// TwinCAT 3 PLC project EtherCatDevice
// Title: EtherCatDevice
// Company: NewEngineer
// Author: https://github.com/phucpha
// ProjectVersion: 0.0.0.2
// Description: this is library use for Device conmunicate by EtherCat without requrire special license.
// ProgramVersion: 3.1.4024.0
// libraries:
//   Tc2_Math, * (Beckhoff Automation GmbH)
//   Tc2_Standard, * (Beckhoff Automation GmbH)
//   Tc2_System, * (Beckhoff Automation GmbH)
//   Tc3_Module, * (Beckhoff Automation GmbH)
//   VisuDialogs, * (System)
//   VisuSymbols,3.5.10.0,System
// project tree:
//   DUTs/Robots/Mitsubishi/CR800/EtherCAT Registers/ ST_CR800EthercatData.TcDUT (not stored)
//   DUTs/Robots/Mitsubishi/CR800/ E_CR800Error.TcDUT (not stored), ST_CR800UserDefinedArea.TcDUT (not stored)
//   DUTs/Robots/Mitsubishi/CR800/StateMachine/ E_CR800State.TcDUT (not stored), E_CR800StateAborting.TcDUT (not stored), E_CR800StateCommandExchange.TcDUT (not stored), E_CR800StateCyclePausing.TcDUT (not stored), E_CR800StateCycleStopping.TcDUT (not stored), E_CR800StateDoingRequest.TcDUT (not stored), E_CR800StateHoming.TcDUT (not stored), E_CR800StateInitializing.TcDUT (not stored), E_CR800StateSendPosition.TcDUT (not stored)
//   DUTs/Robots/Mitsubishi/ E_RobotActions.TcDUT (not stored), E_RobotSystemActions.TcDUT (not stored)
//   DUTs/Visu/ ST_VisuCtrlRobotFrame.TcDUT
//   / GlobalTextList.TcGTLO, PlcTask.TcTTO, Visualization Manager.TcVMO (not stored)
//   POUs/Robots/Mitsubishi/ FB_CR800EtherCAT.TcPOU (not stored), I_CR800EtherCAT.TcIO (not stored)
//   Version/ Global_Version.TcGVL
//   VISUs/Image Polls/ IPRobots.TcIPO (not stored)
//   VISUs/Pages/ PageManualRobots.TcVIS
//   VISUs/Single/ SingleRobot.TcVIS
//   VISUs/Text Lists/ TL_ModeSwitchState.TcTLO, TL_SingleRobotState.TcTLO
// real-time tasks:
//   TASK PlcTask: cycle T#10ms, priority 20, ADS port 350

CONFIGURATION EtherCatDevice
    RESOURCE PLC ON TwinCAT3
        TASK PlcTask(INTERVAL := T#10ms, PRIORITY := 20);
    END_RESOURCE
END_CONFIGURATION

// ---- DUTs/Visu/ST_VisuCtrlRobotFrame.TcDUT
TYPE ST_VisuCtrlRobotFrame :
STRUCT
	sName 						: STRING := 'Unknown';
	btnInit						: BOOL;				(*  *)
	btnAbort					: BOOL;				(*  *)
	btnErrorReset				: BOOL;				(*  *)
	btnControllerReset			: BOOL;				(*  *)
	btnBatteryReset				: BOOL;				(*  *)
	btnGoHome 					: BOOL;				(*  *)
	btnDoAction	 				: BOOL;				(*  *)
	btnUpdateRecipes			: BOOL;				(*  *)
	btnGoAuto 					: BOOL;				(*  *)
	btnCyclePause				: BOOL;				(*  *)
	btnCycleStop				: BOOL;				(*  *)
	btnRestoreCycle 			: BOOL;				(*  *)
	btnRestoreAuto	 			: BOOL;				(*  *)
	btnModeSwitch	 			: BOOL;				(*  *)
	bModeSwitchButtonDisabled	: BOOL;
	
	bError						: BOOL;				(*  *)
	bInit						: BOOL;	
	bPowerOn					: BOOL;	
	bBatteryLow					: BOOL;	
	bIsHomed					: BOOL;
	bServoOn					: BOOL;				(*  *)
	bServoOff 					: BOOL;
	bStarted					: BOOL;
	bStopped					: BOOL;				(*  *)
	bPaused						: BOOL;
	bUninitialized				: BOOL;
	bDoAction					: BOOL;
	bAutoButtonDisable			: BOOL;	
	bActionButtonDisable		: BOOL;	
	bHomeButtonDisable 			: BOOL;
	bPausingButtonDisable 		: BOOL;
	bRestoreCycleButtonDisable  : BOOL;
	bStoppingButtonDisable	    : BOOL;
	bRestoreAutoButtonDisable   : BOOL;
	bInitButtonDisable			: BOOL;
	bModeSwitchState			: BOOL;
	
	sErrorDescription			: STRING;			(*  *)
	iActionNumber				: UINT := 51;		(*  *)
	iOverride					: USINT := 100;
	sStateDescription			: STRING;			(*  *)
	
	sRobotImage					: STRING;			(*  *)
	eRobotState					: E_CR800State;		(*  *)
END_STRUCT
END_TYPE

// ---- Version/Global_Version.TcGVL
{attribute 'TcGenerated'}
{attribute 'no-analysis'}
{attribute 'linkalways'}
// This function has been automatically generated from the project information.
VAR_GLOBAL CONSTANT
	{attribute 'const_non_replaced'}
	stLibVersion_EtherCatDevice : ST_LibVersion := (iMajor := 0, iMinor := 0, iBuild := 0, iRevision := 2, nFlags := 0, sVersion := '0.0.0.2');
END_VAR

// ---- GlobalTextList.TcGTLO
TEXTLIST GlobalTextList
  224 = '%2d'
  331 = '%d'
  976 = '%s'
  2051 = '/'
  887 = 'Abort'
  3798 = 'Action number:'
  427 = 'Auto mode'
  2272 = 'Battery low'
  662 = 'Battery reset'
  1072 = 'Commands'
  1156 = 'Controller'
  2043 = 'Cycle pause'
  3558 = 'Cycle restore'
  1468 = 'Error'
  1738 = 'Error: %s'
  66 = 'Go home'
  1505 = 'Homed'
  371 = 'Initialize'
  1488 = 'Initialized'
  729 = 'Mode switch'
  1606 = 'Next'
  725 = 'Paused'
  731 = 'Powered on'
  1825 = 'Previous'
  316 = 'Program'
  3075 = 'Reset'
  951 = 'Robots'
  2402 = 'Servo off'
  772 = 'Servo on'
  450 = 'Start'
  3789 = 'Started'
  1037 = 'State: %s'
  895 = 'Status'
  1093 = 'Stopped'
END_TEXTLIST

// ---- VISUs/Pages/PageManualRobots.TcVIS
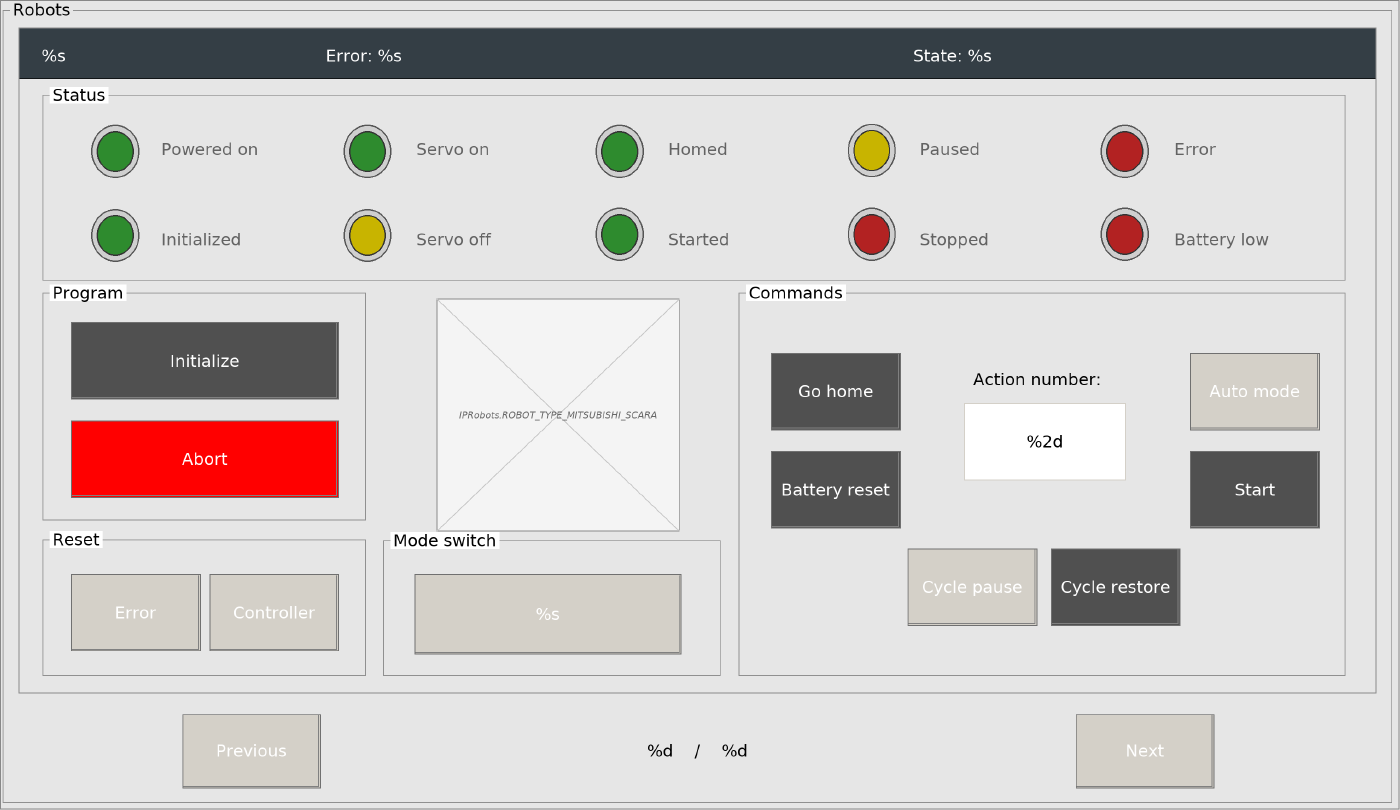
VISUALIZATION PageManualRobots  // 1520x880
VAR_IN_OUT
	btnPrevious			: BOOL;
	btnNext				: BOOL;
	bPreviousInvisible	: BOOL;
	bNextInvisible		: BOOL;
	stRobotEmpty		: ARRAY[1..1] OF BOOL;
	stRobot				: ARRAY[1..1] OF ST_VisuCtrlRobotFrame;
	iRobotSelectedPageIndex	: USINT;
	iRobotTotalPageIndex 	: USINT;
	
END_VAR
    GroupBox (3,3 1508x869), "Robots"
        Button (195,773 150x80), "Previous", invisible if: bPreviousInvisible
            tap btnPrevious
        Button (1165,773 150x80), "Next", invisible if: bNextInvisible
            tap btnNext
        Frame (17,27 1474x723), invisible if: stRobotEmpty[1]
            shows SingleRobot(stRobot := stRobot[1])
        Rectangle (689,788 130x50), "/"
        Rectangle (689,788 50x50), "%d", text variable: iRobotSelectedPageIndex+1
        Rectangle (770,788 50x50), "%d", text variable: iRobotTotalPageIndex+1
END_VISUALIZATION

// ---- VISUs/Single/SingleRobot.TcVIS
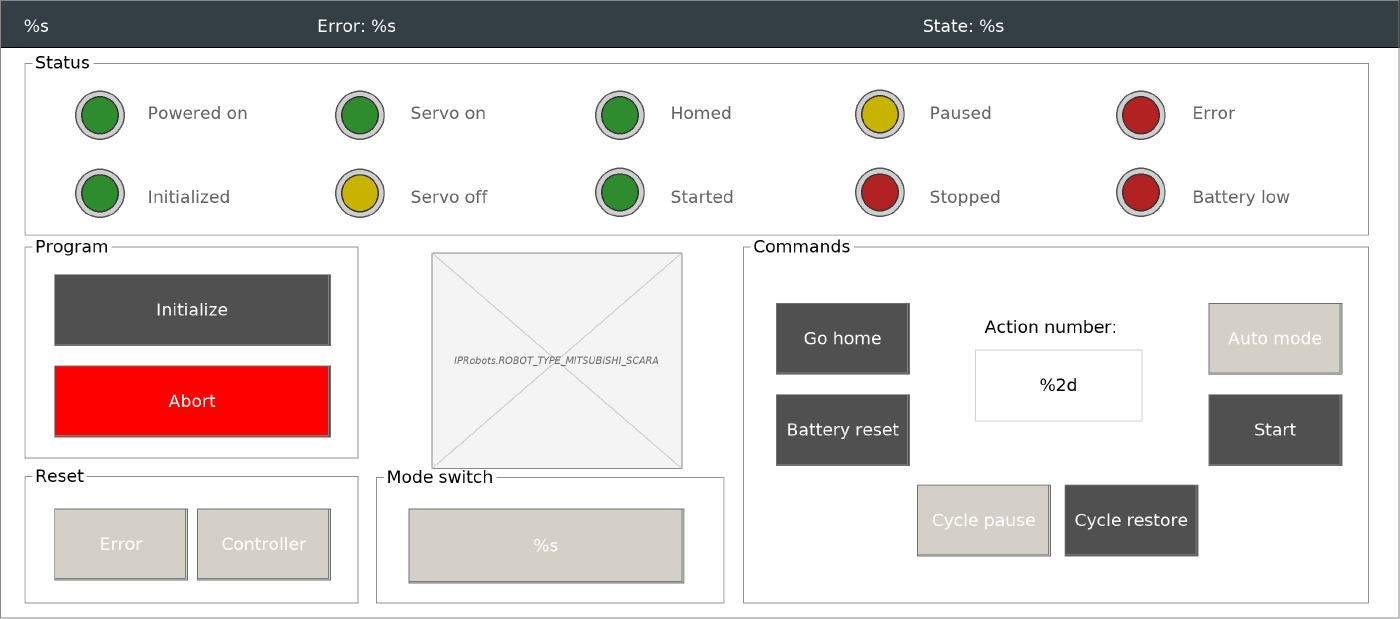
VISUALIZATION SingleRobot  // 1470x650
VAR_IN_OUT
	stRobot		: ST_VisuCtrlRobotFrame;
END_VAR
    Rectangle (0,0 1470x50)
    Textfield (22,10 296x35), "%s", text variable: stRobot.sName
    Textfield (966,10 498x35), "State: %s", text list: 'TL_SingleRobotState', text index: stRobot.eRobotState
    Textfield (330,10 628x35), "Error: %s", text variable: stRobot.sErrorDescription
    Image (453,265 263x227), image: IPRobots.ROBOT_TYPE_MITSUBISHI_SCARA
        p84334746: stRobot.sRobotImage
    GroupBox (26,58 1411x189), "Status"
        Lamp1 (595,33 60x60), variable: stRobot.bIsHomed, style: Lamp-Lamp1-Green
        Lamp1 (595,114 60x60), variable: stRobot.bStarted, style: Lamp-Lamp1-Green
        Rectangle (675,37 150x48), "Homed"
        Rectangle (675,125 150x48), "Started"
        Lamp1 (1142,114 60x60), variable: stRobot.bBatteryLow, style: Lamp-Lamp1-Red
        Rectangle (1223,125 150x48), "Battery low"
        Lamp1 (1142,33 60x60), variable: stRobot.bError, style: Lamp-Lamp1-Red
        Rectangle (1223,37 150x48), "Error"
        Lamp1 (49,33 60x60), variable: stRobot.bPowerOn, style: Lamp-Lamp1-Green
        Lamp1 (49,115 60x60), variable: stRobot.bInit, style: Lamp-Lamp1-Green
        Rectangle (126,37 150x48), "Powered on"
        Rectangle (126,125 150x48), "Initialized"
        Rectangle (402,37 150x48), "Servo on"
        Rectangle (402,125 150x48), "Servo off"
        Lamp1 (322,33 60x60), variable: stRobot.bServoOn, style: Lamp-Lamp1-Green
        Lamp1 (322,115 60x60), variable: stRobot.bServoOff, style: Lamp-Lamp1-Yellow
        Rectangle (947,37 150x48), "Paused"
        Rectangle (947,125 150x48), "Stopped"
        Lamp1 (868,32 60x60), variable: stRobot.bPaused, style: Lamp-Lamp1-Yellow
        Lamp1 (868,114 60x60), variable: stRobot.bStopped, style: Lamp-Lamp1-Red
    GroupBox (26,251 350x230), "Program"
        Button (31,37 290x75), "Initialize", input disabled if: stRobot.bInitButtonDisable
            tap stRobot.btnInit
        Button (31,133 290x75), "Abort", input disabled if: stRobot.bUninitialized
            tap stRobot.btnAbort
    GroupBox (26,492 350x141), "Reset"
        Button (31,42 140x75), "Error"
            tap stRobot.btnErrorReset
        Button (181,42 140x75), "Controller"
            tap stRobot.btnControllerReset
    GroupBox (780,251 657x382), "Commands"
        Button (489,163 140x75), "Start", input disabled if: stRobot.bActionButtonDisable
            tap stRobot.btnDoAction
        Button (35,67 140x75), "Go home", input disabled if: stRobot.bHomeButtonDisable
            tap stRobot.btnGoHome
        Button (489,67 140x75), "Auto mode", input disabled if: stRobot.bAutoButtonDisable
            tap stRobot.btnGoAuto
        Button (35,163 140x75), "Battery reset", input disabled if: stRobot.bAutoButtonDisable
        Rectangle (251,80 160x25), "Action number:"
        Button (338,258 140x75), "Cycle restore", input disabled if: stRobot.bRestoreCycleButtonDisable
            tap stRobot.btnRestoreCycle
        Button (183,258 140x75), "Cycle pause", input disabled if: stRobot.bPausingButtonDisable
            tap stRobot.btnCyclePause
        Textfield (244,116 175x75), "%2d", text variable: stRobot.iActionNumber, input disabled if: stRobot.bActionButtonDisable
            OnMouseClick: write the text variable via VisuDialogs.Numpad, min 13, max 100
    GroupBox (395,493 365x140), "Mode switch", invisible if: stRobot.bModeSwitchButtonDisabled
        Button (34,41 289x78), "%s", input disabled if: stRobot.bInit, text list: 'TL_ModeSwitchState', text index: stRobot.bModeSwitchState
            toggle stRobot.btnModeSwitch
END_VISUALIZATION

// ---- VISUs/Text Lists/TL_ModeSwitchState.TcTLO
TEXTLIST TL_ModeSwitchState
  0 = 'Auto'
  1 = 'Manual'
   = ''
END_TEXTLIST

// ---- VISUs/Text Lists/TL_SingleRobotState.TcTLO
TEXTLIST TL_SingleRobotState
  0 = 'Uninitialized\t'
  10 = 'Initializing'
  20 = 'Ready initialized'
  30 = 'Idle- not homed'
  40 = 'Going home'
  50 = 'Home done'
  60 = 'Idle homed'
  70 = 'Updating recipes'
  80 = 'Updating recipes done'
  100 = 'Going auto'
  110 = 'Going auto done'
  120 = 'Idle auto'
  130 = 'Doing action'
  140 = 'Doing action done'
  200 = 'Cycle stopping'
  210 = 'Cycle stopping done'
  220 = 'Idle auto paused'
  230 = 'Auto restoring'
  240 = 'Auto restoring done'
  300 = 'Cycle pausing'
  310 = 'Cycle pausing done'
  320 = 'Idle cycle paused'
  330 = 'Cycle restoring'
  340 = 'Cycle restoring done'
  500 = 'Reset'
  510 = 'Reset done'
  -10 = 'In external error'
  -20 = 'Aborting'
   = ''
END_TEXTLIST
